{attribute 'pack_mode':='1'}
TYPE AbortToteRequestParams :
STRUCT
   source_id : ModelIdentifier;
   target_id: ModelIdentifier;
END_STRUCT
END_TYPE

(* stored: Version 1.1.0.1, ProductVersion 3.1.4024.12
   DUT AbortToteRequestParams: Id {95488daf-5cbb-4552-bdc5-118075193300} *)
